// TIA Portal project "Akroh-Naaimachine V1.0" (V16)

(* hardware
DEVICE "S71500/ET200MP station_1"  S7-1500 station
   slot 0: "Rail_0"  Rack  6ES7 590-1***0-0AA0
   slot 1: "PLC_1"  CPU 1512C-1 PN  6ES7 512-1CK01-0AB0  V2.8
      slot 3: "CPU display_1"  6ES7591-1AA00-0AA0
      slot 32768: "PROFINET interface_1"  X1
         slot 32769: "Port_1"  X1 P1
         slot 32770: "Port_2"  X1 P2
      slot 34817: "Virtual CP interface port_1"  Virtual CP interface port  Virtual CP interface port
DEVICE "SINAMICS S_1"  AcxSinamics.Device.2x.S210
   slot 0: "Drive_1"  S210 PN  6SL3210-5HB10-4xFx  V5.2
      slot 1: "PROFINET interface"  PROFINET
      slot 3: " Ethernet commissioning interface"  LAN
   slot 0: "Drive control"  S210 PN
      slot 200: "Power Module_1"  Drive control  6SL3210-5HB10-4xFx
      slot 300: "Encoder evaluation_1"  Drive control  1FK2103-4AG0x-xDxx
      slot 400: "Measuring system_1"  Drive control  1FK2103-4AG0x-xDxx
      slot 1000: "Motor_1"  Drive control  1FK2103-4AG0x-xDxx
DEVICE "HMI_1"  KTP700 Basic PN
   slot 0: "HMI_1"  KTP700 Basic PN  6AV2 123-2GB03-0AX0  14.0.0.0
   slot 1: "HMI_RT_1"  KTP700 Basic PN  6AV2 123-2GB03-0AX0  14.0.0.0
   slot 5: "HMI_1.IE_CP_1"  PROFINET Interface  14.0.0.0
      slot 1: "PROFINET Interface_1"  PROFINET Interface
         slot 1: "Port_1"  Port
*)

// ===== PLC "PLC_1"  CPU 1512C-1 PN =====

VAR_GLOBAL   // PLC tag table "Default tag table"
   "PositioningAxis_1_Actor_Interface_AddressIn" AT %I256.0 : "PD_TEL105_IN";
   "S_LineairG_Links" AT %I12.0 : Bool;
   "S_LineairG_Rechts" AT %I12.1 : Bool;
   "S_Grijper_Open" AT %I12.2 : Bool;
   "S_Grijper_Dicht" AT %I12.3 : Bool;
   "S_Cilinder_In" AT %I12.4 : Bool;
   "S_Cilinder_Uit" AT %I12.5 : Bool;
   "S_Schalm_1" AT %I12.6 : Bool;
   "S_Schalm_2" AT %I12.7 : Bool;
   "Start_Knop" AT %I10.0 : Bool;
   "Stop_Knop" AT %I10.1 : Bool;
   "Reset_Knop" AT %I10.2 : Bool;
   "Noodstop_OK" AT %I10.3 : Bool;
   "S_Wiel_Laag" AT %I13.0 : Bool;
   "S_Band" AT %I13.1 : Bool;
   "PositioningAxis_1_Actor_Interface_AddressOut" AT %Q256.0 : "PD_TEL105_OUT";
   "Q_Motor_Links" AT %Q6.0 : Bool;
   "Q_Motor_Rechts" AT %Q6.1 : Bool;
   "Q_LineairA_Links" AT %Q6.2 : Bool;
   "Q_LineairA_Rechts" AT %Q6.3 : Bool;
   "Q_Grijper_Open" AT %Q6.6 : Bool;
   "Q_Cilinder_Uit" AT %Q6.7 : Bool;
   "Q_Wiel_Laag" AT %Q6.4 : Bool;
   "Naaimachine_Klem" AT %Q5.0 : Bool;
   "Naaimachine_Start" AT %Q5.1 : Bool;
   "Naaimachine_Reserve" AT %Q5.2 : Bool;
   "Reset_Noodstop" AT %Q4.0 : Bool;
   "Signaal_LampGroen" AT %Q4.1 : Bool;
   "Signaal_LampOranje" AT %Q4.2 : Bool;
   "Signaal_LampRood" AT %Q4.3 : Bool;
   "Signaal_LampBlauw" AT %Q4.4 : Bool;
   "Signaal_Buzzer" AT %Q4.5 : Bool;
   "Q_Wiel_Hoog(1)" AT %Q6.5 : Bool;
   "Noodstop" AT %I10.4 : Bool;
   "test" AT %I10.5 : Bool;
END_VAR

DATA_BLOCK "Block_1_DB"   // DB11
{ S7_Optimized_Access := 'TRUE' }
VERSION : 0.1
// stored: InstanceOfName Block_1
"Block_1"
BEGIN
END_DATA_BLOCK

DATA_BLOCK "Block_1_DB_1"   // DB17
{ S7_Optimized_Access := 'TRUE' }
VERSION : 0.1
// stored: InstanceOfName Block_1
"Block_1"
BEGIN
END_DATA_BLOCK

DATA_BLOCK "Servo_FB_DB"   // DB28
{ S7_Optimized_Access := 'TRUE' }
VERSION : 0.1
// stored: InstanceOfName Servo_FB
"Servo_FB"
BEGIN
END_DATA_BLOCK

DATA_BLOCK "Eindstation_DB"   // DB29
{ S7_Optimized_Access := 'TRUE' }
VERSION : 0.1
// stored: InstanceOfName Eindstation
"Eindstation"
BEGIN
END_DATA_BLOCK

DATA_BLOCK "ComunicationDB"   // DB30
{ S7_Optimized_Access := 'TRUE' }
VERSION : 0.1
   VAR RETAIN
      Relative_Done : Bool;
   END_VAR
   VAR
      Band_Gemaakt : Bool;
   END_VAR
   VAR RETAIN
      StopSR : Bool;
   END_VAR
BEGIN
END_DATA_BLOCK

DATA_BLOCK "HMI_DB"   // DB32
{ S7_Optimized_Access := 'TRUE' }
VERSION : 0.1
   VAR
      Power_Error : Bool;
      Power_Error_1 : Word;
      Reset_Error : Bool;
      Reset_Error_1 : Word;
      Home_Error : Bool;
      Home_Error_1 : Word;
      Halt_Error : Bool;
      Halt_Error_1 : Word;
      Absolute_Error : Bool;
      Absolute_Error_1 : Word;
      Relative_Error : Bool;
      Relative_Error_1 : Word;
      Velocity_Error : Bool;
      Velocity_Error_1 : Word;
      Jogg_Error : Bool;
      Jogg_Error_1 : Word;
      Stop_Error : Bool;
      Stop_Error_1 : Word;
      ProcesStatus : Int;
      HMI_Driver_Enable : Bool;
   END_VAR
   VAR RETAIN
      Banden_Real_Counter : Int;
      Banden_Totaal_Counter : LInt;
      Banden_Hoeveelheid_Counter : Int := 30;
   END_VAR
   VAR
      Reset_Banden_Totaal : Bool;
   END_VAR
   VAR RETAIN
      SpoelVervangen : Bool;
   END_VAR
   VAR
      Counter_Banden_voldaan : Bool;
   END_VAR
   VAR RETAIN
      Relative_Speed : Int := 800;
      Velocity_Speed : Int := 500;
      Relative_Move_Schalm : Int := 430;
   END_VAR
   VAR
      PowerStatus : Bool;
   END_VAR
BEGIN
END_DATA_BLOCK

// folder: System blocks/Program resources

DATA_BLOCK "IEC_Timer_0_DB"   // DB1
{ S7_Optimized_Access := 'TRUE' }
AUTHOR : Simatic
FAMILY : IEC
NAME : IEC_TMR
VERSION : 1.0
// stored: InstanceOfName IEC_TIMER
"IEC_TIMER"
BEGIN
END_DATA_BLOCK

DATA_BLOCK "IEC_Timer_0_DB_15"   // DB31
{ S7_Optimized_Access := 'TRUE' }
AUTHOR : Simatic
FAMILY : IEC
NAME : IEC_TMR
VERSION : 1.0
// stored: InstanceOfName IEC_TIMER
"IEC_TIMER"
BEGIN
END_DATA_BLOCK

DATA_BLOCK "IEC_Counter_0_DB"   // DB33
{ S7_Optimized_Access := 'TRUE' }
AUTHOR : Simatic
FAMILY : IEC
NAME : CNTR
VERSION : 1.0
// stored: InstanceOfName IEC_COUNTER
"IEC_COUNTER"
BEGIN
END_DATA_BLOCK

DATA_BLOCK "IEC_Counter_0_DB_1"   // DB34
{ S7_Optimized_Access := 'TRUE' }
AUTHOR : SIMATIC
FAMILY : IEC
NAME : LCNTR
VERSION : 1.2
// stored: InstanceOfName IEC_LCOUNTER
"IEC_LCOUNTER"
BEGIN
END_DATA_BLOCK

DATA_BLOCK "IEC_Timer_0_DB_17"   // DB36
{ S7_Optimized_Access := 'TRUE' }
AUTHOR : Simatic
FAMILY : IEC
NAME : IEC_TMR
VERSION : 1.0
// stored: InstanceOfName IEC_TIMER
"IEC_TIMER"
BEGIN
END_DATA_BLOCK

DATA_BLOCK "IEC_Timer_0_DB_20"   // DB39
{ S7_Optimized_Access := 'TRUE' }
AUTHOR : Simatic
FAMILY : IEC
NAME : IEC_TMR
VERSION : 1.0
// stored: InstanceOfName IEC_TIMER
"IEC_TIMER"
BEGIN
END_DATA_BLOCK

DATA_BLOCK "IEC_Timer_0_DB_21"   // DB40
{ S7_Optimized_Access := 'TRUE' }
AUTHOR : Simatic
FAMILY : IEC
NAME : IEC_TMR
VERSION : 1.0
// stored: InstanceOfName IEC_TIMER
"IEC_TIMER"
BEGIN
END_DATA_BLOCK

// folder: (top level)

DATA_BLOCK "SynchronousAxis_1"   // DB18, Motion_DB
{ S7_Optimized_Access := 'TRUE' }
AUTHOR : SIMATIC
FAMILY : MC_1500
VERSION : 5.0
// stored: InstanceOfName TO_SynchronousAxis
"TO_SynchronousAxis"
BEGIN
END_DATA_BLOCK

FUNCTION_BLOCK "Block_1"   // FB1, LAD
{ S7_Optimized_Access := 'TRUE' }
VERSION : 0.1
BEGIN
END_FUNCTION_BLOCK

FUNCTION_BLOCK "Servo_FB"   // FB2, LAD
TITLE = Servo Control
{ S7_Optimized_Access := 'TRUE' }
VERSION : 0.1
   VAR_INPUT
      Enable : Bool;
      Reset : Bool;
      Ack_Technology_Alarms : Bool;
      Set_Home : Bool;
      Halt : Bool;
      Move_Absolute : Bool;
      Absolute_Speed : LReal;
      Absolute_Position : LReal;
      Move_Relative : Bool;
      Relative_Distance : LReal;
      Relative_Speed : LReal;
      Move_Velocity : Bool;
      Velocity_Speed : LReal;
      Direction_Velocity : Int;
      Jog_Forward : Bool;
      Jog_Backward : Bool;
      Jog_Speed : LReal;
      Stop : Bool;
   END_VAR
   VAR_OUTPUT
      Power_Status : Bool;
      Error : Bool;
      ErrorID : Word;
      Reset_Done : Bool;
      Reset_Aborted : Bool;
      Home_Done : Bool;
      Home_Aborted : Bool;
      Halt_Done : Bool;
      Halt_Aborted : Bool;
      Absolute_Position_Reached : Bool;
      Absolute_Position_Aborted : Bool;
      Relative_Move_Done : Bool;
      Relative_Move_Aborted : Bool;
      In_Velocity : Bool;
      Velocity_Aborted : Bool;
      Jog_Aborted : Bool;
      Stopped : Bool;
      Stop_Aborted : Bool;
   END_VAR
BEGIN

REGION Network 1: Power
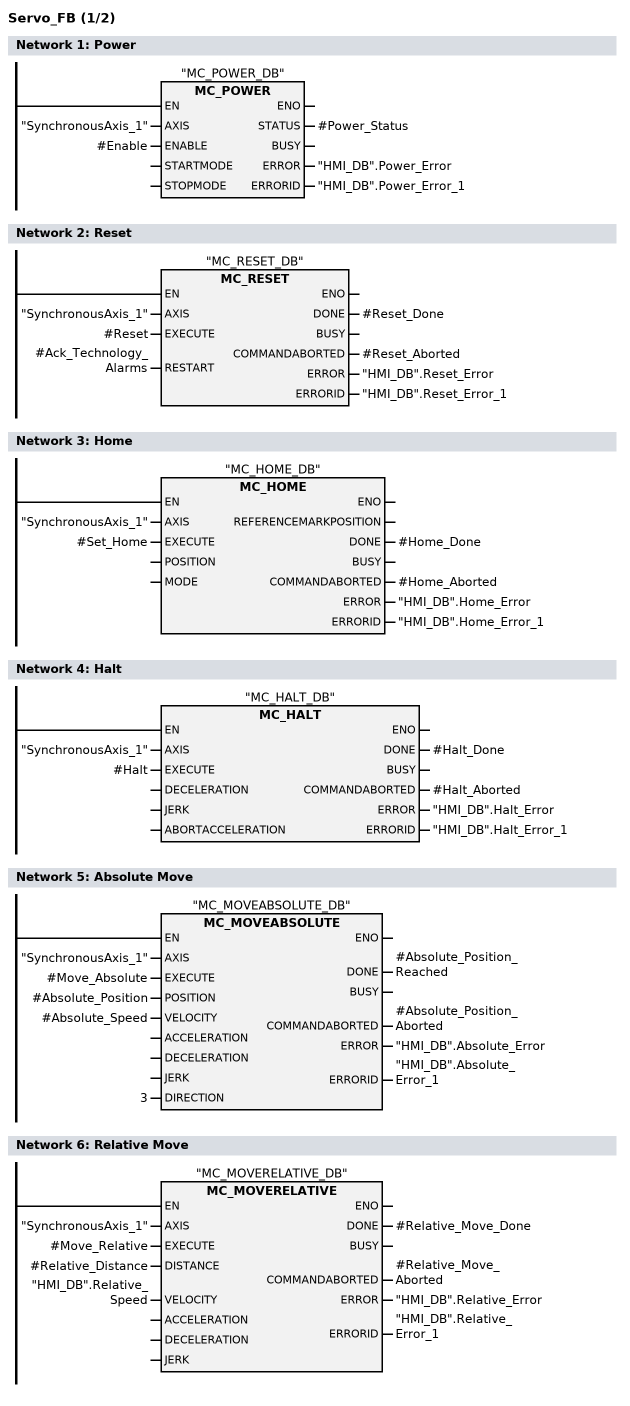
   "MC_POWER_DB"(Axis := "SynchronousAxis_1",   // MC_POWER
                 Enable := #Enable,
                 Status => #Power_Status,
                 Error => "HMI_DB".Power_Error,
                 ErrorId => "HMI_DB".Power_Error_1);
END_REGION

REGION Network 2: Reset
   "MC_RESET_DB"(Axis := "SynchronousAxis_1",   // MC_RESET
                 Execute := #Reset,
                 Restart := #Ack_Technology_Alarms,
                 Done => #Reset_Done,
                 CommandAborted => #Reset_Aborted,
                 Error => "HMI_DB".Reset_Error,
                 ErrorId => "HMI_DB".Reset_Error_1);
END_REGION

REGION Network 3: Home
   "MC_HOME_DB"(Axis := "SynchronousAxis_1",   // MC_HOME
                Execute := #Set_Home,
                Done => #Home_Done,
                CommandAborted => #Home_Aborted,
                Error => "HMI_DB".Home_Error,
                ErrorId => "HMI_DB".Home_Error_1);
END_REGION

REGION Network 4: Halt
   "MC_HALT_DB"(Axis := "SynchronousAxis_1",   // MC_HALT
                Execute := #Halt,
                Done => #Halt_Done,
                CommandAborted => #Halt_Aborted,
                Error => "HMI_DB".Halt_Error,
                ErrorId => "HMI_DB".Halt_Error_1);
END_REGION

REGION Network 5: Absolute Move
   "MC_MOVEABSOLUTE_DB"(Axis := "SynchronousAxis_1",   // MC_MOVEABSOLUTE
                        Execute := #Move_Absolute,
                        Position := #Absolute_Position,
                        Velocity := #Absolute_Speed,
                        Direction := 3,
                        Done => #Absolute_Position_Reached,
                        CommandAborted => #Absolute_Position_Aborted,
                        Error => "HMI_DB".Absolute_Error,
                        ErrorId => "HMI_DB".Absolute_Error_1);
END_REGION

REGION Network 6: Relative Move
   "MC_MOVERELATIVE_DB"(Axis := "SynchronousAxis_1",   // MC_MOVERELATIVE
                        Execute := #Move_Relative,
                        Distance := #Relative_Distance,
                        Velocity := "HMI_DB".Relative_Speed,
                        Done => #Relative_Move_Done,
                        CommandAborted => #Relative_Move_Aborted,
                        Error => "HMI_DB".Relative_Error,
                        ErrorId => "HMI_DB".Relative_Error_1);
END_REGION

REGION Network 7: Velocity
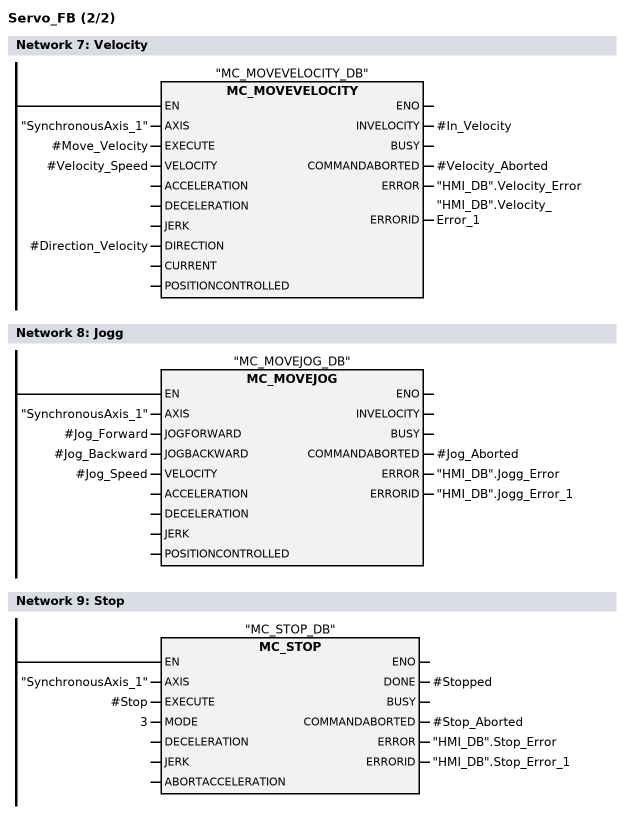
   "MC_MOVEVELOCITY_DB"(Axis := "SynchronousAxis_1",   // MC_MOVEVELOCITY
                        Execute := #Move_Velocity,
                        Velocity := #Velocity_Speed,
                        Direction := #Direction_Velocity,
                        InVelocity => #In_Velocity,
                        CommandAborted => #Velocity_Aborted,
                        Error => "HMI_DB".Velocity_Error,
                        ErrorId => "HMI_DB".Velocity_Error_1);
END_REGION

REGION Network 8: Jogg
   "MC_MOVEJOG_DB"(Axis := "SynchronousAxis_1",   // MC_MOVEJOG
                   JogForward := #Jog_Forward,
                   JogBackward := #Jog_Backward,
                   Velocity := #Jog_Speed,
                   CommandAborted => #Jog_Aborted,
                   Error => "HMI_DB".Jogg_Error,
                   ErrorId => "HMI_DB".Jogg_Error_1);
END_REGION

REGION Network 9: Stop
   "MC_STOP_DB"(Axis := "SynchronousAxis_1",   // MC_STOP
                Execute := #Stop,
                Mode := 3,
                Done => #Stopped,
                CommandAborted => #Stop_Aborted,
                Error => "HMI_DB".Stop_Error,
                ErrorId => "HMI_DB".Stop_Error_1);
END_REGION
END_FUNCTION_BLOCK

FUNCTION_BLOCK "Eindstation"   // FB3, SCL
{ S7_Optimized_Access := 'TRUE' }
VERSION : 0.1
   VAR_INPUT
      Reset : Bool;
      Stop : Bool;
      Start : Bool;
      Sensor_Cilinder_In : Bool;
      Sensor_Cilinder_Uit : Bool;
      Sensor_Gripper_Open : Bool;
      Sensor_Gripper_Dicht : Bool;
      Sensor_Geleider_Links : Bool;
      Sensor_Geleider_Rechts : Bool;
      Band_Sensor : Bool;
      Relative_Done : Bool;
      NoodStop : Bool;
      Afstand_Schalmen : Int;
      Gewacht : Bool;
   END_VAR
   VAR_OUTPUT
      Cilinder_Uit : Bool := 0;
      Gripper_Open : Bool := 1;
      Motor_Links : Bool := 1;
      Motor_Rechts : Bool := 0;
      Geleider_Links : Bool := 0;
      Geleider_Rechts : Bool := 1;
      Ready : Bool := 0;
      Move_Velocity : Bool := 0;
      Move_Relative : Bool := 0;
      Relative_Afstand : Int;
      NaaiPoten_Beneden : Bool := 0;
      Start_Naaien : Bool := 0;
      ffWachten : Bool;
   END_VAR
   VAR
      "Step" : Int := 0;
      PausedStep : Int := 0;
      NextStep : Int := 0;
   END_VAR
   VAR RETAIN
      Genaaid : Bool := 0;
   END_VAR
   VAR
      ProcesStatus : Int;
      Starten : Bool;
      State : Int;
   END_VAR
BEGIN
   // === Start ===
   IF #Start THEN
       #Starten := TRUE;
   END_IF;

   // === RESET Logica ===
   IF #Reset THEN
       #Starten := FALSE;
       #Step := 0;
       #PausedStep := 0;
   END_IF;

   // === STOP/Pauze Logica ===
   //#Step := 0;
   IF #Stop THEN
       #PausedStep := #Step;
       #Step := 99; // Pauzestand

   END_IF;
   // === Noodstop Logica ===
   IF #NoodStop THEN
       #Step := 98; // Noodstopstand

   END_IF;

       // === Normale flow via CASE ===
       CASE #Step OF

               // Stap 0: Initialisatie
           0:
               #State := 0;
               #Gripper_Open := TRUE;
               #Cilinder_Uit := FALSE; 
               #Motor_Rechts := FALSE;
               #Start_Naaien := FALSE;
               #Motor_Links := TRUE;
               #Geleider_Rechts := TRUE;
               #Geleider_Links := FALSE;
               #Move_Relative := FALSE;
               #Move_Velocity := FALSE;
               #Ready := FALSE;
               #ProcesStatus := 0;


               IF #Sensor_Gripper_Open AND #Sensor_Cilinder_In AND #Sensor_Geleider_Rechts AND #Starten THEN
                   #Step := 1;
               END_IF;

           1:
               #State := 1;
               #Cilinder_Uit := TRUE;
               #Gripper_Open := FALSE;
               #Move_Velocity := TRUE;
               #Starten := FALSE;
               #ProcesStatus := 1;

               IF #Sensor_Cilinder_Uit AND #Sensor_Gripper_Dicht THEN
                   #Move_Velocity := FALSE;
                   #Step := 2;
               END_IF;

           2:
               #State := 2;
               #Move_Velocity := TRUE;
               #Motor_Links := FALSE;
               #Motor_Rechts := TRUE;
               #Relative_Afstand := 500;
               #Move_Relative := FALSE;
               #NaaiPoten_Beneden := FALSE;
               #ProcesStatus := 1;


               IF #Band_Sensor THEN
                   #Move_Velocity := FALSE;
                   #Step := 3;
               END_IF;

           3:
               #State := 3;
               #Relative_Afstand := #Afstand_Schalmen;
               #Move_Relative := TRUE;
               #ProcesStatus := 3;
               #ffWachten := FALSE;
               IF #Relative_Done THEN
                   #Move_Relative := FALSE;
                   #Motor_Rechts := False;
                   #Motor_Links := TRUE;
                   #Relative_Afstand := -107;
                   #Step := 4;
               END_IF;
           4:
               #State := 4;
               #ffWachten := TRUE;
               #Move_Relative := TRUE;
               //#Relative_Afstand := -118;


               IF #Gewacht THEN
                   #ffWachten := FALSE;
                   #Gripper_Open := TRUE;
                   #Ready := TRUE;
                   #Step := 11;
               END_IF;

           11:
               #State := 4;
               #ffWachten := TRUE;
               //#Move_Relative := TRUE;

               IF #Gewacht THEN

                   #Step := 5;
               END_IF;

           5:
               #State := 5;
               //#Gripper_Open := TRUE;
               #ffWachten := FALSE;
               #Geleider_Rechts := FALSE;
               #Geleider_Links := TRUE;
               #NaaiPoten_Beneden := FALSE;
               #ProcesStatus := 5;


               IF #Sensor_Geleider_Links AND #Relative_Done THEN
                   #Step := 6;
               END_IF;

           6:
               #State := 6;
               IF #Relative_Done THEN
                   #NaaiPoten_Beneden := TRUE;
                   #ProcesStatus := 6;
                   #ffWachten := TRUE;
               END_IF;
               IF #Gewacht THEN
                   #NaaiPoten_Beneden := FALSE;
                   #ffWachten := FALSE;
                   #Step := 7;
               END_IF;
           7:
               #State := 7;
               #Motor_Links := FALSE;
               #Cilinder_Uit := FALSE;
               #Motor_Rechts := TRUE;
               #Geleider_Links := FALSE;

               #Genaaid := FALSE;


               IF  #Sensor_Cilinder_In THEN
                   #NaaiPoten_Beneden := FALSE;
                   #Step := 8;
               END_IF;
           8:
               #State := 8;
               #Start_Naaien := TRUE;
               #Geleider_Rechts := TRUE;
               #Move_Relative := FALSE;
               #ProcesStatus := 8;
               "IEC_Timer_0_DB_15".TON(IN:= #Sensor_Geleider_Rechts,
                                       PT:=T#8s,
                                       Q=>#Genaaid);
               IF #Genaaid THEN
                   //#NaaiPoten_Beneden := TRUE;
                   #Step := 9;
               END_IF;
           9:
               #State := 9;
               #Start_Naaien := FALSE;
               #Genaaid := FALSE;
               #ProcesStatus := 9;
               #Relative_Afstand := 800;
               #Move_Relative := TRUE;

               IF #Relative_Done THEN
                   #Ready := TRUE;
                   #NaaiPoten_Beneden := FALSE;
                   #Step := 10;
               END_IF;
           10:
               #State := 10;
               #Move_Relative := FALSE;
               #Starten := TRUE;
               #Step := 0;
           98:
               #Move_Velocity := FALSE;
               #ProcesStatus := 98;

           99:
               #Move_Velocity := FALSE;
               #ProcesStatus := 99;
               IF #Start THEN
                   #Step := #State;
               END_IF;
       END_CASE;

       // Stapwissel
       //#Step := #NextStep;
   //END_IF;
END_FUNCTION_BLOCK

FUNCTION_BLOCK "HMI"   // FB4, LAD
{ S7_Optimized_Access := 'TRUE' }
VERSION : 0.1
BEGIN
END_FUNCTION_BLOCK

ORGANIZATION_BLOCK "Main"   // OB1, LAD, ProgramCycle
TITLE = "Main Program Sweep (Cycle)"
{ S7_Optimized_Access := 'TRUE' }
VERSION : 0.1
   VAR_INPUT
      Initial_Call : Bool;   // Initial call of this OB
      Remanence : Bool;   // =True, if remanent data are available
   END_VAR
   VAR_TEMP
      ENDSchalTrue : Bool;
      Puls : Int;
      ResetPuls : Bool;
      Velocity_move : Bool;
      Move_Relative : Bool;
      Relative_Afstand : Int;
      "SR lampRood" : Bool;
      Noodstop_SR : Bool;
      Naaien : Bool;
   END_VAR
BEGIN

REGION Network 1: Fuctie machine
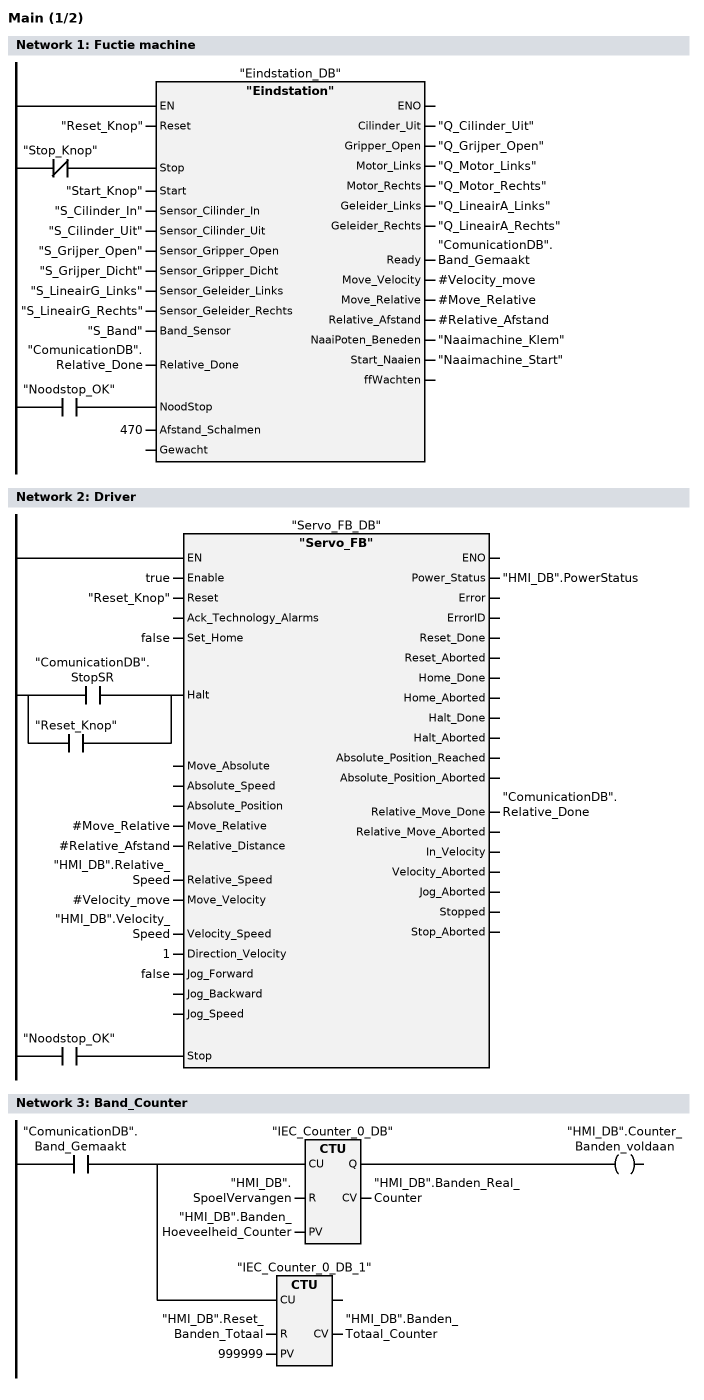
   RUNG wire#powerrail
      "Eindstation_DB"(Stop := wire#w1, NoodStop := wire#w2, Reset := "Reset_Knop", Start := "Start_Knop", Sensor_Cilinder_In := "S_Cilinder_In", Sensor_Cilinder_Uit := "S_Cilinder_Uit", Sensor_Gripper_Open := "S_Grijper_Open", Sensor_Gripper_Dicht := "S_Grijper_Dicht", Sensor_Geleider_Links := "S_LineairG_Links", Sensor_Geleider_Rechts := "S_LineairG_Rechts", Band_Sensor := "S_Band", Relative_Done := "ComunicationDB".Relative_Done, Afstand_Schalmen := 470, Gewacht :=, Cilinder_Uit => "Q_Cilinder_Uit", Gripper_Open => "Q_Grijper_Open", Motor_Links => "Q_Motor_Links", Motor_Rechts => "Q_Motor_Rechts", Geleider_Links => "Q_LineairA_Links", Geleider_Rechts => "Q_LineairA_Rechts", Ready => "ComunicationDB".Band_Gemaakt, Move_Velocity => #Velocity_move, Move_Relative => #Move_Relative, Relative_Afstand => #Relative_Afstand, NaaiPoten_Beneden => "Naaimachine_Klem", Start_Naaien => "Naaimachine_Start", ffWachten =>)
   END_RUNG
   RUNG wire#powerrail
      I_Contact( "Stop_Knop" )
   END_RUNG wire#w1
   RUNG wire#powerrail
      Contact( "Noodstop_OK" )
   END_RUNG wire#w2
   // the same network as SCL:
   "Eindstation_DB"(Reset := "Reset_Knop",   // "Eindstation"
                    Stop := NOT "Stop_Knop",
                    Start := "Start_Knop",
                    Sensor_Cilinder_In := "S_Cilinder_In",
                    Sensor_Cilinder_Uit := "S_Cilinder_Uit",
                    Sensor_Gripper_Open := "S_Grijper_Open",
                    Sensor_Gripper_Dicht := "S_Grijper_Dicht",
                    Sensor_Geleider_Links := "S_LineairG_Links",
                    Sensor_Geleider_Rechts := "S_LineairG_Rechts",
                    Band_Sensor := "S_Band",
                    Relative_Done := "ComunicationDB".Relative_Done,
                    NoodStop := "Noodstop_OK",
                    Afstand_Schalmen := 470,
                    Cilinder_Uit => "Q_Cilinder_Uit",
                    Gripper_Open => "Q_Grijper_Open",
                    Motor_Links => "Q_Motor_Links",
                    Motor_Rechts => "Q_Motor_Rechts",
                    Geleider_Links => "Q_LineairA_Links",
                    Geleider_Rechts => "Q_LineairA_Rechts",
                    Ready => "ComunicationDB".Band_Gemaakt,
                    Move_Velocity => #Velocity_move,
                    Move_Relative => #Move_Relative,
                    Relative_Afstand => #Relative_Afstand,
                    NaaiPoten_Beneden => "Naaimachine_Klem",
                    Start_Naaien => "Naaimachine_Start");
END_REGION

REGION Network 2: Driver
   RUNG wire#powerrail
      "Servo_FB_DB"(Halt := wire#w1, Stop := wire#w2, Enable := true, Reset := "Reset_Knop", Ack_Technology_Alarms :=, Set_Home := false, Move_Absolute :=, Absolute_Speed :=, Absolute_Position :=, Move_Relative := #Move_Relative, Relative_Distance := #Relative_Afstand, Relative_Speed := "HMI_DB".Relative_Speed, Move_Velocity := #Velocity_move, Velocity_Speed := "HMI_DB".Velocity_Speed, Direction_Velocity := 1, Jog_Forward := false, Jog_Backward :=, Jog_Speed :=, Power_Status => "HMI_DB".PowerStatus, Error =>, ErrorID =>, Reset_Done =>, Reset_Aborted =>, Home_Done =>, Home_Aborted =>, Halt_Done =>, Halt_Aborted =>, Absolute_Position_Reached =>, Absolute_Position_Aborted =>, Relative_Move_Done => "ComunicationDB".Relative_Done, Relative_Move_Aborted =>, In_Velocity =>, Velocity_Aborted =>, Jog_Aborted =>, Stopped =>, Stop_Aborted =>)
   END_RUNG
   RUNG wire#powerrail
      Contact( "ComunicationDB".StopSR )
   END_RUNG wire#w1
   RUNG wire#powerrail
      Contact( "Reset_Knop" )
   END_RUNG wire#w1
   RUNG wire#powerrail
      Contact( "Noodstop_OK" )
   END_RUNG wire#w2
   // the same network as SCL:
   "Servo_FB_DB"(Enable := true,   // "Servo_FB"
                 Reset := "Reset_Knop",
                 Set_Home := false,
                 Halt := "ComunicationDB".StopSR OR "Reset_Knop",
                 Move_Relative := #Move_Relative,
                 Relative_Distance := #Relative_Afstand,
                 Relative_Speed := "HMI_DB".Relative_Speed,
                 Move_Velocity := #Velocity_move,
                 Velocity_Speed := "HMI_DB".Velocity_Speed,
                 Direction_Velocity := 1,
                 Jog_Forward := false,
                 Stop := "Noodstop_OK",
                 Power_Status => "HMI_DB".PowerStatus,
                 Relative_Move_Done => "ComunicationDB".Relative_Done);
END_REGION

REGION Network 3: Band_Counter
   "IEC_Counter_0_DB".CTU(CU := "ComunicationDB".Band_Gemaakt,
                          R := "HMI_DB".SpoelVervangen,
                          PV := "HMI_DB".Banden_Hoeveelheid_Counter,
                          CV => "HMI_DB".Banden_Real_Counter);
   "HMI_DB".Counter_Banden_voldaan := "IEC_Counter_0_DB".Q;
   "IEC_Counter_0_DB_1".CTU(CU := "ComunicationDB".Band_Gemaakt,
                           R := "HMI_DB".Reset_Banden_Totaal,
                           PV := 999999,
                           CV => "HMI_DB".Banden_Totaal_Counter);
END_REGION

REGION Network 4: Signaal toren
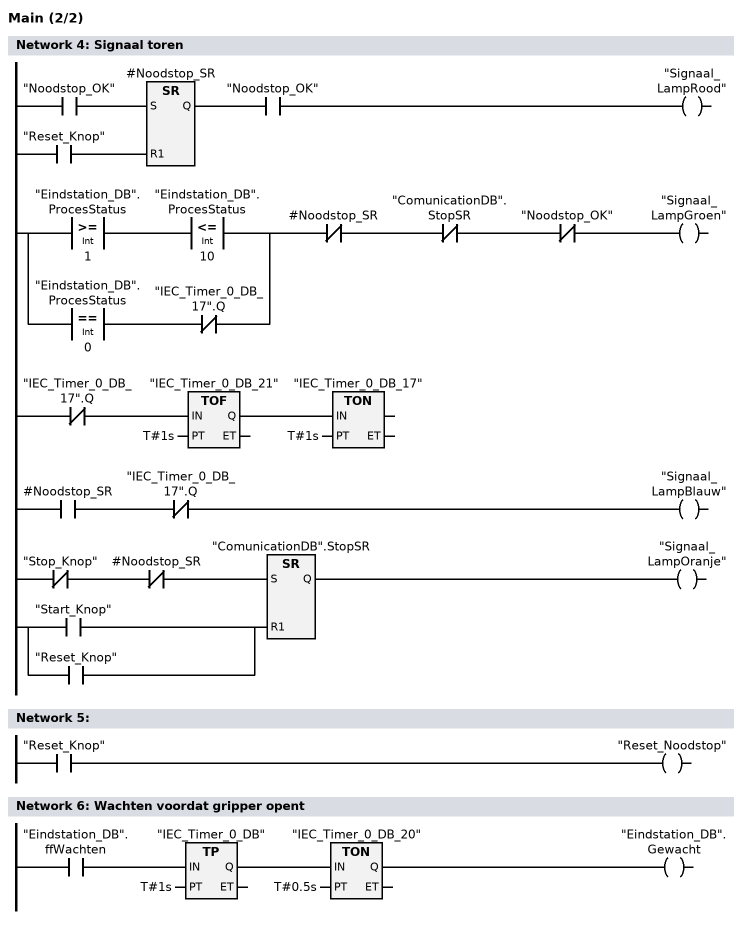
   IF "Noodstop_OK" THEN
       #Noodstop_SR := TRUE;   // SR flip-flop
   END_IF;
   IF "Reset_Knop" THEN #Noodstop_SR := FALSE; END_IF;
   "Signaal_LampRood" := #Noodstop_SR AND "Noodstop_OK";
   "Signaal_LampGroen" := ((("Eindstation_DB".ProcesStatus >= 1) AND ("Eindstation_DB".ProcesStatus <= 10)) OR (("Eindstation_DB".ProcesStatus = 0) AND NOT "IEC_Timer_0_DB_17".Q)) AND NOT #Noodstop_SR AND NOT "ComunicationDB".StopSR AND NOT "Noodstop_OK";
   "IEC_Timer_0_DB_21".TOF(IN := NOT "IEC_Timer_0_DB_17".Q, PT := T#1s);
   "IEC_Timer_0_DB_17".TON(IN := "IEC_Timer_0_DB_21".Q, PT := T#1s);
   "Signaal_LampBlauw" := #Noodstop_SR AND NOT "IEC_Timer_0_DB_17".Q;
   IF NOT "Stop_Knop" AND NOT #Noodstop_SR THEN
       "ComunicationDB".StopSR := TRUE;   // SR flip-flop
   END_IF;
   IF "Start_Knop" OR "Reset_Knop" THEN "ComunicationDB".StopSR := FALSE; END_IF;
   "Signaal_LampOranje" := "ComunicationDB".StopSR;
END_REGION

REGION Network 5
   RUNG wire#powerrail
      Contact( "Reset_Knop" )
      Coil( "Reset_Noodstop" )
   END_RUNG
   // the same network as SCL:
   "Reset_Noodstop" := "Reset_Knop";
END_REGION

REGION Network 6: Wachten voordat gripper opent
   "IEC_Timer_0_DB".TP(IN := "Eindstation_DB".ffWachten, PT := T#1s);
   "IEC_Timer_0_DB_20".TON(IN := "IEC_Timer_0_DB".Q, PT := T#0.5s);
   "Eindstation_DB".Gewacht := "IEC_Timer_0_DB_20".Q;
END_REGION
END_ORGANIZATION_BLOCK

(* ===== HMI "HMI_RT_1" =====
system functions are stored by id; their names below are inferred from use
connection "HMI_Connection_1": ETHERNET, SMART_S7_1500_OMS

HMI tags "Default tag table"
   "Tag_ScreenNumber" : UInt, internal
   "HMI_DB_Banden_Hoeveelheid_Counter" : Int = PLC HMI_DB.Banden_Hoeveelheid_Counter, 1 s
   "HMI_DB_Banden_Real_Counter" : Int = PLC HMI_DB.Banden_Real_Counter, 1 s
   "HMI_DB_Banden_Totaal_Counter" : LInt = PLC HMI_DB.Banden_Totaal_Counter, 1 s
   "SynchronousAxis_1_Base_Base_StatusDrive_Error" : Bool = PLC SynchronousAxis_1.StatusDrive.Error, 1 s
   "SynchronousAxis_1_Base_Base_StatusDrive_CommunicationOK" : Bool = PLC SynchronousAxis_1.StatusDrive.CommunicationOK, 1 s
   "SynchronousAxis_1_Base_Base_StatusDrive_InOperation" : Bool = PLC SynchronousAxis_1.StatusDrive.InOperation, 1 s
   "SynchronousAxis_1_Base_Base_StatusTorqueData_ActualTorque" : LReal = PLC SynchronousAxis_1.StatusTorqueData.ActualTorque, 1 s
   "SynchronousAxis_1_Base_Base_DynamicLimits_MaxAcceleration" : LReal = PLC SynchronousAxis_1.DynamicLimits.MaxAcceleration, 1 s
   "SynchronousAxis_1_Base_Base_DynamicLimits_MaxDeceleration" : LReal = PLC SynchronousAxis_1.DynamicLimits.MaxDeceleration, 1 s
   "SynchronousAxis_1_Base_Base_DynamicLimits_MaxJerk" : LReal = PLC SynchronousAxis_1.DynamicLimits.MaxJerk, 1 s
   "SynchronousAxis_1_Base_Base_DynamicLimits_MaxVelocity" : LReal = PLC SynchronousAxis_1.DynamicLimits.MaxVelocity, 1 s
   "SynchronousAxis_1_Base_Clamping_PositionTolerance" : LReal = PLC SynchronousAxis_1.Clamping.PositionTolerance, 1 s
   "Servo_FB_DB_Halt" : Bool = PLC Servo_FB_DB.Halt, 1 s
   "Servo_FB_DB_Jog_Forward" : Bool = PLC Servo_FB_DB.Jog_Forward, 1 s
   "Servo_FB_DB_Jog_Backward" : Bool = PLC Servo_FB_DB.Jog_Backward, 1 s
   "Servo_FB_DB_Direction_Velocity" : Int = PLC Servo_FB_DB.Direction_Velocity, 1 s
   "Servo_FB_DB_Jog_Speed" : LReal = PLC Servo_FB_DB.Jog_Speed, 1 s
   "Start_Knop" : Bool = PLC Start_Knop AT %I10.0, 1 s
   "Stop_Knop" : Bool = PLC Stop_Knop AT %I10.1, 1 s
   "Reset_Knop" : Bool = PLC Reset_Knop AT %I10.2, 1 s
   "HMI_DB_ProcesStatus" : Int = PLC HMI_DB.ProcesStatus, 1 s
   "Eindstation_DB_ProcesStatus" : Int = PLC Eindstation_DB.ProcesStatus, 1 s
   "S_Band_1" : Bool = PLC S_Wiel_Laag AT %I13.0, 1 s
   "S_Schalm_1" : Bool = PLC S_Schalm_1 AT %I12.6, 1 s
   "S_Schalm_2" : Bool = PLC S_Schalm_2 AT %I12.7, 1 s

Template "Template_1" 800x480
   DateTimeField "HmiScreenItemData" at 695,25 size 105x25
   DateTimeField "HmiScreenItemData_1" at 695,0 size 105x25
   GraphicView "Logo" at 0,0 size 137x51; Picture "Logo of HMI_1"

screen "Root screen" 800x480, template "Template_1"
   on GenerateScreen: SetTag("Tag_ScreenNumber", 1)
   Rectangle "Rectangle_2" at 53,61 size 325x151
      Appearance <- "Eindstation_DB_ProcesStatus"
   TextField "Text field_1" at 65,70 size 157x29; Text 'Proces Status:'
   TextField "Text field_2" at 65,260 size 227x29; Text 'Proces Driver Status:'
   TextField "Text field_3" at 522,70 size 181x29; Text 'Spoel Informatie'
   TextField "Text field_4" at 503,130 size 213x27; Text 'Spoel verwisselen na:'
   TextField "Text field_5" at 503,207 size 238x27; Text 'Huidige Banden gedaan:'
   TextField "Text field_6" at 503,290 size 224x27; Text 'Totale Banden gedaan:'
   IOField "I/O field_1" at 527,167 size 96x32; FormatPattern 99; Unit  
      ProcessValue <- "HMI_DB_Banden_Hoeveelheid_Counter"
   TextField "Text field_7" at 629,170 size 76x27; Text 'Banden'
   IOField "I/O field_2" at 527,250 size 96x32; FormatPattern 99; Unit  
      ProcessValue <- "HMI_DB_Banden_Real_Counter"
   TextField "Text field_8" at 629,253 size 76x27; Text 'Banden'
   IOField "I/O field_3" at 527,333 size 96x32; FormatPattern 99999999; Unit  
      ProcessValue <- "HMI_DB_Banden_Totaal_Counter"
   TextField "Text field_9" at 629,336 size 76x27; Text 'Banden'
   Rectangle "Rectangle_8" at 53,298 size 108x33
      Appearance <- "SynchronousAxis_1_Base_Base_StatusDrive_Error"
   Rectangle "Rectangle_9" at 161,298 size 107x33
      Appearance <- "SynchronousAxis_1_Base_Base_StatusDrive_CommunicationOK"
   Rectangle "Rectangle_10" at 268,298 size 110x33
      Appearance <- "SynchronousAxis_1_Base_Base_StatusDrive_InOperation"
   TextField "Text field_10" at 84,304 size 46x23; Text 'Error'
   TextField "Text field_11" at 159,304 size 110x22; Text 'Communicatie'
   TextField "Text field_12" at 272,304 size 100x22; Text 'In Operation'
   TextField "Text field_13" at 65,349 size 16x23; Text 'Text'
   IOField "I/O field_4" at 241,349 size 110x32; FormatPattern 999.99; Unit  Nm
      ProcessValue <- "SynchronousAxis_1_Base_Base_StatusTorqueData_ActualTorque"
   TextField "Text field_14" at 73,351 size 158x29; Text 'Actual Torque:'
   Button "Button_1" at 326,254 size 51x43; TextOff 'Text'; PictureOff "instellingen"
      on Press: ActivateScreen("Driver_Instelling", 0)
   Button "Button_2" at 5,432 size 50x45; TextOff 'Text'; PictureOff "NavigateHome_KTP700_Basic_PN_TR"
      on Press: ActivateScreen("Root screen", 0)
   Button "Button_4" at 325,432 size 50x45; TextOff 'Text'; PictureOff "Play"
      on Press: function_b14e0dd5("Start_Knop", 0)
   Button "Button_5" at 383,432 size 50x45; TextOff 'Text'; PictureOff "pause"
      on Press: function_b14e0dd5("Stop_Knop", 0)
   Button "Button_6" at 441,432 size 50x45; TextOff 'Text'; PictureOff "reset"
      on Press: function_b14e0dd5("Reset_Knop", 0)
   TextField "Text field_15" at 101,121 size 230x43; Text 'Begin Posities'
      Visibility <- "Eindstation_DB_ProcesStatus"
   TextField "Text field_16" at 76,121 size 285x43; Text 'Wachten op Band'
      Visibility <- "Eindstation_DB_ProcesStatus"
   TextField "Text field_17" at 60,122 size 311x43; Text 'Band Gedetecteerd'
      Visibility <- "Eindstation_DB_ProcesStatus"
   TextField "Text field_18" at 65,126 size 303x37; Text 'Band naar Naaipositie'
      Visibility <- "Eindstation_DB_ProcesStatus"
   TextField "Text field_19" at 102,120 size 247x43; Text 'Band Klemmen'
      Visibility <- "Eindstation_DB_ProcesStatus"
   TextField "Text field_20" at 151,122 size 117x43; Text 'Naaien'
      Visibility <- "Eindstation_DB_ProcesStatus"
   TextField "Text field_21" at 95,122 size 262x43; Text 'Band Uitwerpen'
      Visibility <- "Eindstation_DB_ProcesStatus"
   TextField "Text field_22" at 158,121 size 130x43; Text 'Gestopt'
      Visibility <- "Eindstation_DB_ProcesStatus"
   TextField "Text field_23" at 131,122 size 159x43; Text 'Noodstop'
      Visibility <- "Eindstation_DB_ProcesStatus"
   Rectangle "Rectangle_11" at 53,175 size 167x37
      Appearance <- "S_Schalm_1"
   Rectangle "Rectangle_12" at 219,175 size 159x37
      Appearance <- "S_Schalm_2"
   TextField "Text field_24" at 99,182 size 78x23; Text 'Schalm 1'
   TextField "Text field_25" at 258,182 size 78x23; Text 'Schalm 2'

screen "Driver_Instelling" 800x480, template "Template_1"
   IOField "I/O field_1" at 200,124 size 96x32; FormatPattern 999999
      ProcessValue <- "SynchronousAxis_1_Base_Base_DynamicLimits_MaxAcceleration"
   TextField "Text field_1" at 32,129 size 152x23; Text 'Max Acceleration:'
   IOField "I/O field_2" at 200,171 size 96x32; FormatPattern 999999
      ProcessValue <- "SynchronousAxis_1_Base_Base_DynamicLimits_MaxDeceleration"
   TextField "Text field_2" at 32,176 size 154x23; Text 'Max Deceleration:'
   IOField "I/O field_3" at 200,218 size 96x32; FormatPattern 999999
      ProcessValue <- "SynchronousAxis_1_Base_Base_DynamicLimits_MaxJerk"
   TextField "Text field_3" at 32,223 size 85x23; Text 'Max Jerk:'
   IOField "I/O field_4" at 200,265 size 96x32; FormatPattern 999999
      ProcessValue <- "SynchronousAxis_1_Base_Base_DynamicLimits_MaxVelocity"
   TextField "Text field_4" at 32,270 size 115x23; Text 'Max Velocity:'
   IOField "I/O field_5" at 200,312 size 96x32; FormatPattern 99999.999
      ProcessValue <- "SynchronousAxis_1_Base_Clamping_PositionTolerance"
   TextField "Text field_5" at 32,317 size 163x23; Text 'Position Tolerance:'
   Button "Button_1" at 402,239 size 109x32; TextOff 'Backward'
      on Press: SetTag("Servo_FB_DB_Jog_Backward", 1)
      on Release: SetTag("Servo_FB_DB_Jog_Backward", 0)
   Button "Button_2" at 523,239 size 96x32; TextOff 'Halt'
      on Press: InvertBit("Servo_FB_DB_Halt")
   Button "Button_3" at 630,239 size 114x32; TextOff 'Froward'
      on Press: SetTag("Servo_FB_DB_Jog_Forward", 1)
      on Release: SetTag("Servo_FB_DB_Jog_Forward", 0)
   TextField "Text field_6" at 378,165 size 55x29; Text 'Jogg'
   TextField "Text field_7" at 449,197 size 102x23; Text 'Jogg speed:'
   IOField "I/O field_6" at 574,194 size 96x32; FormatPattern 999999
      ProcessValue <- "Servo_FB_DB_Jog_Speed"
   Button "Button_4" at 5,432 size 50x45; TextOff 'Text'; PictureOff "NavigateHome_KTP700_Basic_PN_TR"
      on Press: ActivateScreen("Root screen", 0)
   IOField "I/O field_7" at 607,333 size 110x32; FormatPattern 999.99; Unit  Nm
      ProcessValue <- "SynchronousAxis_1_Base_Base_StatusTorqueData_ActualTorque"
   TextField "Text field_14" at 439,335 size 158x29; Text 'Actual Torque:'
*)